// TwinCAT 3 PLC project EcSlavePLC
// ProgramVersion: 3.1.4026.23
// libraries:
//   Tc2_ControllerToolbox, * (Beckhoff Automation GmbH)
//   Tc2_Standard, * (Beckhoff Automation GmbH)
//   Tc2_System, * (Beckhoff Automation GmbH)
// project tree:
//   / PlcTask.TcTTO
//   POUs/ MAIN.TcPOU
// (motion and I/O tree: see PLC project plc1)
// real-time tasks:
//   TASK Plc1Task: cycle T#10ms, priority 10, ADS port 350
//   TASK Plc2Task: cycle T#10ms, priority 14, ADS port 351
//   TASK EcSlaveTask: cycle T#10ms, priority 3, ADS port 352
// variable links:

CONFIGURATION EcSlavePLC
    RESOURCE PLC ON TwinCAT3
        TASK PlcTask(INTERVAL := T#10ms, PRIORITY := 3);
        PROGRAM MAIN WITH PlcTask : MAIN;
    END_RESOURCE
END_CONFIGURATION

// ---- POUs/MAIN.TcPOU
PROGRAM MAIN
VAR
	Counter	AT%Q*:UINT;
	fbSinWave	:FB_CTRL_SIGNAL_GENERATOR;
	Param: ST_CTRL_SIGNAL_GENERATOR_PARAMS := (tCtrlCycleTime := TIME#10ms, tTaskCycleTime := TIME#10ms, tCylceDuration := TIME#2s0ms, fAmplitude := 1000);
END_VAR

fbSinWave( 
	eMode:=E_CTRL_MODE.eCTRL_MODE_ACTIVE , 
	stParams:=Param );
	
	
Counter:=TO_UINT(fbSinWave.fOut);

END_PROGRAM
